(* IEC 61131-3 sources: actuators/src/PositionControl, 4 files *)

(* ---- PositionBehavior.st ---- *)
USING System.Timer;

NAMESPACE Simatic.Ax.Actuators
    /// Enumeration defining position behavior for actuator control.
    /// Input: None.
    /// Returns: ActiveHold - keeps output active, SelfHold - sets output to false.
    TYPE
        PositionBehavior : (ActiveHold, SelfHold) := SelfHold; // SelfHold --> Set Q to false, ActiveHold --> Keep Q on True
    END_TYPE
END_NAMESPACE

(* ---- itfPositionControl.st ---- *)
USING System.Timer;

NAMESPACE Simatic.Ax.Actuators
    /// Interface for defining methods to control actuator positions.
    /// Input: Various control commands.
    /// Returns: BOOL indicating success/state of the operation.
    INTERFACE itfPositionControl
        /// Sets the actuator position to active.
        /// Input: None.
        /// Returns: BOOL indicating the operation result.
        METHOD Set : BOOL
        END_METHOD

        /// Holds the actuator position based on the configured behavior.
        /// Input: None.
        /// Returns: BOOL indicating the operation result.
        METHOD Hold : BOOL
        END_METHOD

        /// Resets the actuator position to inactive.
        /// Input: None.
        /// Returns: BOOL indicating the operation result.
        METHOD Reset : BOOL
        END_METHOD
    END_INTERFACE
END_NAMESPACE

(* ---- NullPositionControl.st ---- *)
USING System.Timer;

NAMESPACE Simatic.Ax.Actuators
    /// Internal class providing a dummy implementation of the itfPositionControl interface.
    /// Input: None.
    /// Returns: Default BOOL values for all methods (no actual functionality).
    CLASS INTERNAL NullPositionControl
        IMPLEMENTS itfPositionControl

        /// Dummy implementation of Set method.
        /// Input: None.
        /// Returns: Default BOOL value.
        METHOD PUBLIC Set : BOOL
            ;
        END_METHOD

        /// Dummy implementation of Reset method.
        /// Input: None.
        /// Returns: Default BOOL value.
        METHOD PUBLIC Reset : BOOL
            ;
        END_METHOD

        /// Dummy implementation of Hold method.
        /// Input: None.
        /// Returns: Default BOOL value.
        METHOD PUBLIC Hold : BOOL
            ;
        END_METHOD
    END_CLASS
END_NAMESPACE

(* ---- PositionControl.st ---- *)
USING System.Timer;

NAMESPACE Simatic.Ax.Actuators
    /// Class providing control logic for actuator positions.
    /// Input: Position control commands via Set, Reset, Hold methods.
    /// Returns: Position state and cyclic output signal.
    CLASS PositionControl
        IMPLEMENTS itfPositionControl

        // Public variables
        VAR PUBLIC
            /// Defines the behavior of the actuator position: ActiveHold or SelfHold.
            Behavior : PositionBehavior;
        END_VAR

        // Protected variables
        VAR PROTECTED
            /// Internal state of the actuator position.
            _q : BOOL;
        END_VAR

        /// Writes the cyclic output signal.
        /// Input: None.
        /// Returns: Q - Output signal representing the actuator state.
        METHOD PUBLIC WriteCyclic
            VAR_OUTPUT
                /// Output signal representing the actuator state.
                Q : BOOL;
            END_VAR
            Q := _q;
        END_METHOD

        /// Sets the actuator position to active.
        /// Input: None.
        /// Returns: BOOL indicating the operation result.
        METHOD PUBLIC Set : BOOL
            _q := TRUE;
            Set := _q;
        END_METHOD

        /// Resets the actuator position to inactive.
        /// Input: None.
        /// Returns: BOOL indicating the operation result.
        METHOD PUBLIC Reset : BOOL
            _q := FALSE;
            Reset := _q;
        END_METHOD

        /// Holds the actuator position based on the configured behavior.
        /// Input: None.
        /// Returns: BOOL indicating the operation result.
        METHOD PUBLIC Hold : BOOL
            IF (Behavior = PositionBehavior#ActiveHold) THEN
                _q := TRUE;
            ELSE
                _q := FALSE;
            END_IF;
            Hold := _q;
        END_METHOD
    END_CLASS
END_NAMESPACE
